(* CoDeSys 2.3 export: FLOWBATCHERSUBSTATUS.EXP *)

(* Data type in ENUM *)
TYPE FlowBatcherSubStatus : (FlowBatcherSubStatusNormal:=0, FlowBatcherSubStatusBatching, FlowBatcherSubStatusPause, FlowBatcherSubStatusRefStopped,
									FlowBatcherSubStatusRefAlarm, FlowBatcherSubStatusConfErr, FlowBatcherSubStatusForbiddenCommand,
									FlowBatcherSubStatusUnknownCommand, FlowBatcherSubStatusBadCommandParameter);
END_TYPE
